FUNCTION_BLOCK fb_eje_reset
VAR_IN_OUT
	var_ref_eje : ref_eje_io;
END_VAR
VAR_INPUT
	in_flg_reset : BOOL;
END_VAR
VAR_OUTPUT
	out_flg_resetDone: BOOL;
END_VAR
VAR

	fbi_ton1: TON;
	var_process: INT;
END_VAR


fbi_ton1(IN:= , PT:=T#100MS , Q=> , ET=> );

IF NOT in_flg_reset THEN
	var_process := 0;
END_IF
CASE var_process OF
	0:
		IF in_flg_reset THEN
			var_process := 1;
		END_IF
	1:
		fbi_ton1.IN := FALSE;
		var_process := 2;
	2:	
		fbi_ton1.IN := TRUE;
		var_ref_eje.param.var_mutex := 0;
		var_ref_eje.output.out_flg_ejeVac := FALSE;
		var_ref_eje.output.out_flg_ejeBrk := FALSE;
		IF fbi_ton1.Q THEN
			var_process := 3;
		END_IF
	3:
		out_flg_resetDone := TRUE;
		var_process := 4;
	4:
		out_flg_resetDone := FALSE;
END_CASE

END_FUNCTION_BLOCK

(* stored: Version 1.1.0.1, ProductVersion 3.1.4024.11
   POU fb_eje_reset: Id {be0f5e4d-ba7e-4d5a-bd36-bcbdae64764b}, SpecialFunc None *)
